(* IEC 61131-3 sources: AXOpen/src/components.rexroth.drives/ctrl/src/AxoCtrlxDriveXsc/v_6_x_x (part 3) *)

        ///<summary>
        /// This method  commands a controlled motion of a specified distance relative to the set position at the time of the execution.
        ///</summary>
        VAR INTERNAL
            MC_MoveRelativeExecute_PV					: 	BOOL;				//Execute - previous value
            MC_MoveRelativeErrorID					    : 	DINT;
            MC_MoveRelativeCycle					    : 	ULINT;
            MC_MoveRelativeContinuousUpdate_SV          :   BOOL;
            MC_MoveRelativeDistance_PV                  :   LREAL;
            MC_MoveRelativeVelocity_PV                  :   LREAL;
            MC_MoveRelativeAcceleration_PV              :   LREAL;
            MC_MoveRelativeDeceleration_PV              :   LREAL;
            MC_MoveRelativeJerk_PV                      :   LREAL;
        END_VAR
        METHOD PUBLIC OVERRIDE MC_MoveRelative
            VAR_INPUT
                AxisRef         :   AXOpen.Components.Abstractions.Drives.IAxoAxisReference;
                Execute         :   BOOL;                       //  Start the motion at rising edge
                ContinuousUpdate:   BOOL;                       //  Activate ‘ContinuousUpdate’ - target parameters should be changed during movement
                Distance        :   LREAL;                      //  Relative distance for the motion (in technical unit [u]
                Velocity        :   LREAL;                      //  Value of the maximum ‘Velocity’ (not necessarily reached) [u/s].
                Acceleration    :   LREAL;                      //  Value of the ‘Acceleration’ (always positive) (increasing energy of the motor) [u/s2]
                Deceleration    :   LREAL;                      //  Value of the ‘Deceleration’ (always positive) (decreasing energy of the motor) [u/s2]
                Jerk            :   LREAL;                      //  Value of the ‘Jerk’ [u/s3]
            END_VAR
            VAR_OUTPUT
                Done            :   BOOL;                       // Commanded distance reached
                Busy            :   BOOL;                       // The method is not finished and new output values are to be expected
                Active          :   BOOL;                       // Indicates that the method has control on the axis
                CommandAborted  :   BOOL;                       // ‘Command’ is aborted by another command
                Error           :   BOOL;                       // Signals that an error has occurred within the method
                ErrorID         :   DINT;                       // Error identification
            END_VAR
            VAR
                _AxisReference :  REF_TO AxoCtrlxDriveXscAxisReference;
            END_VAR

            _AxisReference ?= AxisRef;

            IF(_AxisReference = NULL) THEN
                Messenger.Activate(     UINT#1500, eAxoMessageCategory#ProgrammingError);
                DriveStatus.Error.Id := UINT#1500;
                RETURN;
            END_IF;

            IF THIS.AxoMoveRelative_Task.StartTriggered()  THEN
                _AxisReference^.Status.CurrentMotionTaskId := AXOpen.Components.Drives.eAxoMotionTaskId#Axo_MoveRelative;
            END_IF;

            IF Execute AND NOT MC_MoveRelativeExecute_PV AND _State = UINT#0 THEN
                _AxisReference^.Data.Cycle := _AxisReference^.Data.Cycle + ULINT#2;
                MC_MoveRelativeCycle := _AxisReference^.Data.Cycle ;
            END_IF;

            IF Execute THEN
                Messenger.ActivateOnCondition(ULINT#1501, Execute AND Velocity <= 0, eAxoMessageCategory#ProgrammingError);
                Messenger.ActivateOnCondition(ULINT#1502, Execute AND Acceleration <= 0, eAxoMessageCategory#ProgrammingError);
                Messenger.ActivateOnCondition(ULINT#1503, Execute AND Deceleration <= 0, eAxoMessageCategory#ProgrammingError);
                Messenger.ActivateOnCondition(ULINT#1504, Execute AND Jerk <= 0, eAxoMessageCategory#ProgrammingError);

                IF NOT ContinuousUpdate THEN
                    MC_MoveRelativeContinuousUpdate_SV := FALSE;
                END_IF;

                IF _State = UINT#0 THEN
                    Busy := TRUE;
                    Active := TRUE;
                    MC_MoveRelativeErrorID := DINT#0;
                    _AxisReference^.Outputs.SignalControlWord_S_0_0145_0_0.JogPositive := FALSE;
                    _AxisReference^.Outputs.SignalControlWord_S_0_0145_0_0.JogNegative := FALSE;
                    _AxisReference^.Outputs.SignalControlWord_S_0_0145_0_0.HomingControl:= FALSE;
                    _AxisReference^.Outputs.SignalControlWord_S_0_0145_0_0.AbsoluteRelative := TRUE;
                    _AxisReference^.Outputs.SignalControlWord_S_0_0145_0_0.ImmediateChange := TRUE;
                    MC_MoveRelativeContinuousUpdate_SV := ContinuousUpdate;
                    _State := UINT#360;
                    THIS.CallTimers(FALSE);
                END_IF;
                IF _State = UINT#360 THEN
                    IF _infoTimer.output THEN
                        TaskMessenger.Activate( UINT#560, eAxoMessageCategory#Potential);
                        DriveStatus.Error.Id := UINT#560;
                    END_IF;
                    Busy := TRUE;
                    Active := TRUE;
                    IF Velocity > 0 AND Acceleration > 0 AND Deceleration >0 AND Jerk > 0 THEN
                        _AxisReference^.Outputs.CommandPosition_S_0_0282_0_0 :=         TO_DINT(Distance        *   ScalingConstantRequiredPosition);
                        _AxisReference^.Outputs.CommandVelocity_S_0_0259_0_0 :=         TO_DINT(Velocity        *   ScalingConstantRequiredVelocity     * _AxisReference^.Data.OverrideVelocityFactor);
                        _AxisReference^.Outputs.CommandAcceleration_S_0_0260_0_0 :=     TO_DINT(Acceleration    *   ScalingConstantRequiredAcceleration * _AxisReference^.Data.OverrideAccelerationFactor);
                        _AxisReference^.Outputs.CommandDecceleration_S_0_0359_0_0 :=    TO_DINT(Deceleration    *   ScalingConstantRequiredDeceleration * _AxisReference^.Data.OverrideAccelerationFactor);
                        _AxisReference^.Outputs.CommandJerk_S_0_0193_0_0 :=             TO_DINT(Jerk            *   ScalingConstantRequiredJerk         * _AxisReference^.Data.OverrideJerkFactor);
                        MC_MoveRelativeDistance_PV      :=  Distance;
                        MC_MoveRelativeVelocity_PV      :=  Velocity;
                        MC_MoveRelativeAcceleration_PV  :=  Acceleration;
                        MC_MoveRelativeDeceleration_PV  :=  Deceleration;
                        MC_MoveRelativeJerk_PV          :=  Jerk;
                        _State := UINT#361;
                        THIS.CallTimers(FALSE);
                    END_IF;
                END_IF;
                IF _State = UINT#361 THEN
                    IF _infoTimer.output THEN
                        TaskMessenger.Activate( UINT#561, eAxoMessageCategory#Potential);
                        DriveStatus.Error.Id := UINT#561;
                    END_IF;
                    Busy := TRUE;
                    Active := TRUE;
                    _AxisReference^.Outputs.DriveControlWord_S_0_0134_0_0.CommandOperationModeBit0  := FALSE;
                    _AxisReference^.Outputs.DriveControlWord_S_0_0134_0_0.CommandOperationModeBit1  := FALSE;
                    _AxisReference^.Outputs.DriveControlWord_S_0_0134_0_0.CommandOperationModeBit2  := FALSE;
                    IF  NOT _AxisReference^.Inputs.DriveStatusWord_S_0_0135_0_0.ActualOperatingModeBit0 AND
                        NOT _AxisReference^.Inputs.DriveStatusWord_S_0_0135_0_0.ActualOperatingModeBit1 AND
                        NOT _AxisReference^.Inputs.DriveStatusWord_S_0_0135_0_0.ActualOperatingModeBit2 THEN
                        _State := UINT#362;
                        THIS.CallTimers(FALSE);
                    END_IF;
                END_IF;
                IF _State = UINT#362 THEN
                    IF _infoTimer.output THEN
                        TaskMessenger.Activate( UINT#562, eAxoMessageCategory#Potential);
                        DriveStatus.Error.Id := UINT#562;
                    END_IF;
                    Busy := TRUE;
                    Active := TRUE;
                    IF  _AxisReference^.Inputs.DriveStatusWord_S_0_0135_0_0.ReadyForOperationBit0 AND
                        _AxisReference^.Inputs.DriveStatusWord_S_0_0135_0_0.ReadyForOperationBit1 THEN
                       _State := UINT#363;
                        THIS.CallTimers(FALSE);
                    END_IF;
                END_IF;
                IF _State = UINT#363 THEN
                    IF _infoTimer.output THEN
                        TaskMessenger.Activate( UINT#563, eAxoMessageCategory#Potential);
                        DriveStatus.Error.Id := UINT#563;
                    END_IF;
                    Busy := TRUE;
                    Active := TRUE;
                    _AxisReference^.Outputs.DriveControlWord_S_0_0134_0_0.DriveHalt  := TRUE;
                    IF _AxisReference^.Inputs.DriveStatusWord_S_0_0135_0_0.CommandProcessingStatus AND NOT _AxisReference^.Inputs.DriveStatusWord_S_0_0135_0_0.InStandstill  THEN
                       _State := UINT#364;
                        THIS.CallTimers(FALSE);
                    END_IF;
                END_IF;
                //Executing movement
                IF _State = UINT#364 THEN
                    IF _infoTimer.output THEN
                        TaskMessenger.Activate( UINT#564, eAxoMessageCategory#Potential);
                        DriveStatus.Error.Id := UINT#564;
                    END_IF;
                    Busy := TRUE;
                    Active := TRUE;
                    _AxisReference^.Outputs.SignalControlWord_S_0_0145_0_0.AcceptanceOfPositioningCommandValue := NOT _AxisReference^.Outputs.SignalControlWord_S_0_0145_0_0.AcceptanceOfPositioningCommandValue; //_AxisReference^.Outputs.SignalControlWord_S_0_0145_0_0.AcceptanceOfPositioningCommandValue := NOT _AxisReference^.Inputs.SignalStatusWord_S_0_0144_0_0.PositionCommandAck;
                    IF TRUE THEN
                        _State := UINT#365;
                        THIS.CallTimers(FALSE);
                    END_IF;
                END_IF;
                IF _State = UINT#365 THEN
                    IF _infoTimer.output THEN
                        TaskMessenger.Activate( UINT#565, eAxoMessageCategory#Potential);
                        DriveStatus.Error.Id := UINT#565;
                    END_IF;
                    Busy := TRUE;
                    Active := TRUE;
                    IF _AxisReference^.Outputs.SignalControlWord_S_0_0145_0_0.AcceptanceOfPositioningCommandValue = _AxisReference^.Inputs.SignalStatusWord_S_0_0144_0_0.PositionCommandAck THEN
                        _State := UINT#366;
                        THIS.CallTimers(FALSE);
                    END_IF;
                END_IF;
                IF _State = UINT#366 THEN
                    IF _infoTimer.output THEN
                        TaskMessenger.Activate( UINT#566, eAxoMessageCategory#Potential);
                        DriveStatus.Error.Id := UINT#566;
                    END_IF;
                    IF _AxisReference^.Inputs.SignalStatusWord_S_0_0144_0_0.DriveStandstill AND _AxisReference^.Inputs.SignalStatusWord_S_0_0144_0_0.InTargetPosition THEN
                        _State := UINT#367;
                        THIS.CallTimers(FALSE);
                    END_IF;
                END_IF;
                IF _State = UINT#367 THEN
                    Done := TRUE;
                    MC_MoveRelativeCycle := ULINT#0;
                END_IF;
                IF _State = UINT#368 THEN
                    CommandAborted := TRUE; // action handled in parent AxoDrive
                END_IF;
                IF _State = UINT#369 THEN
                    MC_MoveRelativeCycle := ULINT#0;
                    Error := TRUE; // action handled in parent AxoDrive
                END_IF;

                IF _State>=UINT#360 AND _State<UINT#367 THEN
                    IF MC_MoveRelativeContinuousUpdate_SV AND (
                        MC_MoveRelativeDistance_PV      <>  Distance OR
                        MC_MoveRelativeVelocity_PV      <>  Velocity OR
                        MC_MoveRelativeAcceleration_PV  <>  Acceleration OR
                        MC_MoveRelativeDeceleration_PV  <>  Deceleration OR
                        MC_MoveRelativeJerk_PV          <>  Jerk ) THEN
                        IF TRUE THEN
                            _AxisReference^.Outputs.CommandPosition_S_0_0282_0_0 :=         TO_DINT(Distance        *   ScalingConstantRequiredPosition);
                            _AxisReference^.Outputs.CommandVelocity_S_0_0259_0_0 :=         TO_DINT(Velocity        *   ScalingConstantRequiredVelocity     * _AxisReference^.Data.OverrideVelocityFactor);
                            _AxisReference^.Outputs.CommandAcceleration_S_0_0260_0_0 :=     TO_DINT(Acceleration    *   ScalingConstantRequiredAcceleration * _AxisReference^.Data.OverrideAccelerationFactor);
                            _AxisReference^.Outputs.CommandDecceleration_S_0_0359_0_0 :=    TO_DINT(Deceleration    *   ScalingConstantRequiredDeceleration * _AxisReference^.Data.OverrideAccelerationFactor);
                            _AxisReference^.Outputs.CommandJerk_S_0_0193_0_0 :=             TO_DINT(Jerk            *   ScalingConstantRequiredJerk         * _AxisReference^.Data.OverrideJerkFactor);
                            MC_MoveRelativeDistance_PV      :=  Distance;
                            MC_MoveRelativeVelocity_PV      :=  Velocity;
                            MC_MoveRelativeAcceleration_PV  :=  Acceleration;
                            MC_MoveRelativeDeceleration_PV  :=  Deceleration;
                            MC_MoveRelativeJerk_PV          :=  Jerk;
                            _State := UINT#361;
                        END_IF;
                    END_IF;
                    IF NOT _AxisReference^.Inputs.DriveStatusWord_S_0_0135_0_0.ReadyForOperationBit0 OR NOT _AxisReference^.Inputs.DriveStatusWord_S_0_0135_0_0.ReadyForOperationBit1 THEN
                        _State := UINT#368;
                    ELSIF _AxisReference^.Inputs.DriveStatusWord_S_0_0135_0_0.DriveErrorZKL1 OR
                        (_AxisReference^.Inputs.DriveStatusWord_S_0_0135_0_0.WarningZKL2 AND _AxisReference^.Inputs.DiagnosticMessage_S_0_0390_0_0 >= DWORD#16#C00E0000) THEN
                        IF MC_MoveRelativeErrorID = DINT#0 THEN
                            MC_MoveRelativeErrorID := TO_DINT(_AxisReference^.Inputs.DiagnosticMessage_S_0_0390_0_0 AND DWORD#16#000FFFFF);
                        END_IF;
                        _State := UINT#369;
                    ELSIF _AxisReference^.Data.Cycle <> MC_MoveRelativeCycle THEN
                        _AxisReference^.Data.Cycle := _AxisReference^.Data.Cycle - ULINT#1;
                        _State := UINT#368;
                    END_IF;
                END_IF;

                THIS.CallTimers(TRUE,FALSE);
                THIS.AxoMoveRelative_Task.ThrowWhen(_errorTimer.output );
                THIS.AxoMoveRelative_Task.ThrowWhen(THIS.AxoMoveRelative_Task.Duration >= DriveConfig.TaskTimeout AND DriveConfig.TaskTimeout > T#0s ,'<#AxoMoveRelative_Task timeout.#>');
                DriveStatus.Action.Id := _State;
            END_IF;

            IF THIS.AxoMoveRelative_Task.DoneReached() AND _State>=UINT#360 AND _State<=UINT#369 THEN
                _AxisReference^.Status.CurrentMotionTaskId := AXOpen.Components.Drives.eAxoMotionTaskId#Axo_Done;
                MC_MoveRelativeErrorID := DINT#0;
                // MC_MoveRelativeCycle := ULINT#0;
                _State := UINT#0;
            END_IF;

            IF THIS.AxoMoveRelative_Task.RestoreTriggered() AND _State>=UINT#360 AND _State<=UINT#369 THEN
                _AxisReference^.Status.CurrentMotionTaskId := AXOpen.Components.Drives.eAxoMotionTaskId#Axo_None;
                MC_MoveRelativeErrorID := DINT#0;
                MC_MoveRelativeCycle := ULINT#0;
                _State := UINT#0;
            END_IF;
            ErrorID := MC_MoveRelativeErrorID;
            MC_MoveRelativeExecute_PV := Execute;
        END_METHOD

        ///<summary>
        /// This method commands a controlled motion of a specified relative distance additional to the most recent
        /// commanded position in the axis_State ‘DiscreteMotion’. The most recent commanded position may be the result of a
        /// previous MC_MoveAdditive motion which was aborted. If the method is activated in the axis_State ‘ContinuousMotion’, the
        /// specified relative distance is added to the set position at the time of the execution.
        ///</summary>
        VAR INTERNAL
            MC_MoveAdditiveExecute_PV					: 	BOOL;				//Execute - previous value
            MC_MoveAdditiveErrorID					    : 	DINT;
            MC_MoveAdditiveCycle					    : 	ULINT;
            MC_MoveAdditiveContinuousUpdate_SV          :   BOOL;
            MC_MoveAdditiveDistance_PV                  :   LREAL;
            MC_MoveAdditiveVelocity_PV                  :   LREAL;
            MC_MoveAdditiveAcceleration_PV              :   LREAL;
            MC_MoveAdditiveDeceleration_PV              :   LREAL;
            MC_MoveAdditiveJerk_PV                      :   LREAL;
        END_VAR
        METHOD PUBLIC OVERRIDE MC_MoveAdditive
            VAR_INPUT
                AxisRef         :   AXOpen.Components.Abstractions.Drives.IAxoAxisReference;
                Execute         :   BOOL;                       //  Start the motion at rising edge
                ContinuousUpdate:   BOOL;                       //  Activate ‘ContinuousUpdate’ - target parameters should be changed during movement
                Distance        :   LREAL;                      //  Relative distance for the motion (in technical unit [u]
                Velocity        :   LREAL;                      //  Value of the maximum ‘Velocity’ (not necessarily reached) [u/s].
                Acceleration    :   LREAL;                      //  Value of the ‘Acceleration’ (always positive) (increasing energy of the motor) [u/s2]
                Deceleration    :   LREAL;                      //  Value of the ‘Deceleration’ (always positive) (decreasing energy of the motor) [u/s2]
                Jerk            :   LREAL;                      //  Value of the ‘Jerk’ [u/s3]
            END_VAR
            VAR_OUTPUT
                Done            :   BOOL;                       // Commanded distance reached
                Busy            :   BOOL;                       // The method is not finished and new output values are to be expected
                Active          :   BOOL;                       // Indicates that the method has control on the axis
                CommandAborted  :   BOOL;                       // ‘Command’ is aborted by another command
                Error           :   BOOL;                       // Signals that an error has occurred within the method
                ErrorID         :   DINT;                       // Error identification
            END_VAR
            VAR
                _AxisReference :  REF_TO AxoCtrlxDriveXscAxisReference;
            END_VAR

            _AxisReference ?= AxisRef;

            IF(_AxisReference = NULL) THEN
                Messenger.Activate(     UINT#1510, eAxoMessageCategory#ProgrammingError);
                DriveStatus.Error.Id := UINT#1510;
                RETURN;
            END_IF;

            IF Execute AND NOT MC_MoveAdditiveExecute_PV THEN
                _State := UINT#0;  //TODO check if this casues the issue with two move relative movements???
            END_IF;

            IF Execute THEN
                Messenger.ActivateOnCondition(ULINT#1511, Execute AND Velocity <= 0, eAxoMessageCategory#ProgrammingError);
                Messenger.ActivateOnCondition(ULINT#1512, Execute AND Acceleration <= 0, eAxoMessageCategory#ProgrammingError);
                Messenger.ActivateOnCondition(ULINT#1513, Execute AND Deceleration <= 0, eAxoMessageCategory#ProgrammingError);
                Messenger.ActivateOnCondition(ULINT#1514, Execute AND Jerk <= 0, eAxoMessageCategory#ProgrammingError);

                IF NOT ContinuousUpdate THEN
                    MC_MoveAdditiveContinuousUpdate_SV := FALSE;
                END_IF;

                IF _State = UINT#0 THEN
                    Busy := TRUE;
                    Active := TRUE;
                    MC_MoveAdditiveErrorID := DINT#0;
                    _AxisReference^.Outputs.SignalControlWord_S_0_0145_0_0.JogPositive := FALSE;
                    _AxisReference^.Outputs.SignalControlWord_S_0_0145_0_0.JogNegative := FALSE;
                    _AxisReference^.Outputs.SignalControlWord_S_0_0145_0_0.HomingControl:= FALSE;
                    _AxisReference^.Outputs.SignalControlWord_S_0_0145_0_0.ImmediateChange := TRUE;
                    MC_MoveAdditiveContinuousUpdate_SV := ContinuousUpdate;
                    IF Velocity > 0 AND Acceleration > 0 AND Deceleration >0 AND Jerk > 0 THEN
                        MC_MoveAdditiveDistance_PV      :=  Distance;
                        MC_MoveAdditiveVelocity_PV      :=  Velocity;
                        MC_MoveAdditiveAcceleration_PV  :=  Acceleration;
                        MC_MoveAdditiveDeceleration_PV  :=  Deceleration;
                        MC_MoveAdditiveJerk_PV          :=  Jerk;
                        IF _AxisReference^.Status.CurrentMotionTaskId = eAxoMotionTaskId#Axo_MoveAbsolute THEN
                            AxoMoveAbsolute_Task.Abort();
                            _AxisReference^.Outputs.SignalControlWord_S_0_0145_0_0.AbsoluteRelative := FALSE;
                            _AxisReference^.Outputs.CommandPosition_S_0_0282_0_0 :=         TO_DINT((MC_MoveAbsolutePosition_PV + Distance) * ScalingConstantRequiredPosition);
                            _AxisReference^.Outputs.CommandVelocity_S_0_0259_0_0 :=         TO_DINT(Velocity        *   ScalingConstantRequiredVelocity         * _AxisReference^.Data.OverrideVelocityFactor);
                            _AxisReference^.Outputs.CommandAcceleration_S_0_0260_0_0 :=     TO_UINT(Acceleration    *   ScalingConstantRequiredAcceleration     * _AxisReference^.Data.OverrideAccelerationFactor);
                            _AxisReference^.Outputs.CommandDecceleration_S_0_0359_0_0 :=    TO_UINT(Deceleration    *   ScalingConstantRequiredDeceleration     * _AxisReference^.Data.OverrideAccelerationFactor);
                            _AxisReference^.Outputs.CommandJerk_S_0_0193_0_0 :=             TO_DINT(Jerk            *   ScalingConstantRequiredJerk             * _AxisReference^.Data.OverrideJerkFactor);
                        ELSE
                            _AxisReference^.Outputs.SignalControlWord_S_0_0145_0_0.AbsoluteRelative := TRUE;
                            _AxisReference^.Outputs.CommandPosition_S_0_0282_0_0 :=         TO_DINT((Distance)      *   ScalingConstantRequiredPosition);
                            _AxisReference^.Outputs.CommandVelocity_S_0_0259_0_0 :=         TO_DINT(Velocity        *   ScalingConstantRequiredVelocity         * _AxisReference^.Data.OverrideVelocityFactor);
                            _AxisReference^.Outputs.CommandAcceleration_S_0_0260_0_0 :=     TO_UINT(Acceleration    *   ScalingConstantRequiredAcceleration     * _AxisReference^.Data.OverrideAccelerationFactor);
                            _AxisReference^.Outputs.CommandDecceleration_S_0_0359_0_0 :=    TO_UINT(Deceleration    *   ScalingConstantRequiredDeceleration     * _AxisReference^.Data.OverrideAccelerationFactor);
                            _AxisReference^.Outputs.CommandJerk_S_0_0193_0_0 :=             TO_DINT(Jerk            *   ScalingConstantRequiredJerk             * _AxisReference^.Data.OverrideJerkFactor);
                        END_IF;
                        IF _AxisReference^.Status.CurrentMotionTaskId = eAxoMotionTaskId#Axo_MoveRelative THEN
                            AxoMoveRelative_Task.Abort();
                        END_IF;
                        _AxisReference^.Status.CurrentMotionTaskId := eAxoMotionTaskId#Axo_MoveAdditive;
                        _AxisReference^.Data.Cycle := _AxisReference^.Data.Cycle + ULINT#2;
                        MC_MoveAdditiveCycle := _AxisReference^.Data.Cycle ;
                        _State := UINT#371;
                        THIS.CallTimers(FALSE);
                    END_IF;
                END_IF;
                IF _State = UINT#370 THEN
                    _State := UINT#371;
                    THIS.CallTimers(FALSE);
                END_IF;
                IF _State = UINT#371 THEN
                    IF _infoTimer.output THEN
                        TaskMessenger.Activate( UINT#571, eAxoMessageCategory#Potential);
                        DriveStatus.Error.Id := UINT#571;
                    END_IF;
                    Busy := TRUE;
                    Active := TRUE;
                    _AxisReference^.Outputs.DriveControlWord_S_0_0134_0_0.CommandOperationModeBit0  := FALSE;
                    _AxisReference^.Outputs.DriveControlWord_S_0_0134_0_0.CommandOperationModeBit1  := FALSE;
                    _AxisReference^.Outputs.DriveControlWord_S_0_0134_0_0.CommandOperationModeBit2  := FALSE;
                    IF  NOT _AxisReference^.Inputs.DriveStatusWord_S_0_0135_0_0.ActualOperatingModeBit0 AND
                        NOT _AxisReference^.Inputs.DriveStatusWord_S_0_0135_0_0.ActualOperatingModeBit1 AND
                        NOT _AxisReference^.Inputs.DriveStatusWord_S_0_0135_0_0.ActualOperatingModeBit2 THEN
                        _State := UINT#372;
                        THIS.CallTimers(FALSE);
                    END_IF;
                END_IF;
                IF _State = UINT#372 THEN
                    IF _infoTimer.output THEN
                        TaskMessenger.Activate( UINT#572, eAxoMessageCategory#Potential);
                        DriveStatus.Error.Id := UINT#572;
                    END_IF;
                    Busy := TRUE;
                    Active := TRUE;
                    IF  _AxisReference^.Inputs.DriveStatusWord_S_0_0135_0_0.ReadyForOperationBit0 AND
                        _AxisReference^.Inputs.DriveStatusWord_S_0_0135_0_0.ReadyForOperationBit1 THEN
                       _State := UINT#373;
                        THIS.CallTimers(FALSE);
                    END_IF;
                END_IF;
                IF _State = UINT#373 THEN
                    IF _infoTimer.output THEN
                        TaskMessenger.Activate( UINT#573, eAxoMessageCategory#Potential);
                        DriveStatus.Error.Id := UINT#573;
                    END_IF;
                    Busy := TRUE;
                    Active := TRUE;
                    _AxisReference^.Outputs.DriveControlWord_S_0_0134_0_0.DriveHalt  := TRUE;
                    IF _AxisReference^.Inputs.DriveStatusWord_S_0_0135_0_0.CommandProcessingStatus AND NOT _AxisReference^.Inputs.DriveStatusWord_S_0_0135_0_0.InStandstill  THEN
                       _State := UINT#374;
                        THIS.CallTimers(FALSE);
                    END_IF;
                END_IF;
                IF _State = UINT#374 THEN
                    IF _infoTimer.output THEN
                        TaskMessenger.Activate( UINT#574, eAxoMessageCategory#Potential);
                        DriveStatus.Error.Id := UINT#574;
                    END_IF;
                    Busy := TRUE;
                    Active := TRUE;
                    _AxisReference^.Outputs.SignalControlWord_S_0_0145_0_0.AcceptanceOfPositioningCommandValue := NOT _AxisReference^.Outputs.SignalControlWord_S_0_0145_0_0.AcceptanceOfPositioningCommandValue; //_AxisReference^.Outputs.SignalControlWord_S_0_0145_0_0.AcceptanceOfPositioningCommandValue := NOT _AxisReference^.Inputs.SignalStatusWord_S_0_0144_0_0.PositionCommandAck;
                    IF TRUE THEN
                        _State := UINT#375;
                        THIS.CallTimers(FALSE);
                    END_IF;
                END_IF;
                IF _State = UINT#375 THEN
                    IF _infoTimer.output THEN
                        TaskMessenger.Activate( UINT#575, eAxoMessageCategory#Potential);
                        DriveStatus.Error.Id := UINT#575;
                    END_IF;
                    Busy := TRUE;
                    Active := TRUE;
                    IF _AxisReference^.Outputs.SignalControlWord_S_0_0145_0_0.AcceptanceOfPositioningCommandValue = _AxisReference^.Inputs.SignalStatusWord_S_0_0144_0_0.PositionCommandAck THEN
                        _State := UINT#376;
                        THIS.CallTimers(FALSE);
                    END_IF;
                END_IF;
                IF _State = UINT#376 THEN
                    IF _infoTimer.output THEN
                        TaskMessenger.Activate( UINT#576, eAxoMessageCategory#Potential);
                        DriveStatus.Error.Id := UINT#576;
                    END_IF;
                    IF _AxisReference^.Inputs.SignalStatusWord_S_0_0144_0_0.DriveStandstill AND _AxisReference^.Inputs.SignalStatusWord_S_0_0144_0_0.InTargetPosition THEN
                        _State := UINT#377;
                        THIS.CallTimers(FALSE);
                    END_IF;
                END_IF;
                IF _State = UINT#377 THEN
                    Done := TRUE;
                    MC_MoveAdditiveCycle := ULINT#0;
                END_IF;
                IF _State = UINT#378 THEN
                    CommandAborted := TRUE; // action handled in parent AxoDrive
                END_IF;
                IF _State = UINT#379 THEN
                    MC_MoveAdditiveCycle := ULINT#0;
                    Error := TRUE; // action handled in parent AxoDrive
                END_IF;

                IF _State>=UINT#370 AND _State<UINT#377 THEN
                    IF MC_MoveAdditiveContinuousUpdate_SV AND (
                        MC_MoveAdditiveDistance_PV      <>  Distance OR
                        MC_MoveAdditiveVelocity_PV      <>  Velocity OR
                        MC_MoveAdditiveAcceleration_PV  <>  Acceleration OR
                        MC_MoveAdditiveDeceleration_PV  <>  Deceleration OR
                        MC_MoveAdditiveJerk_PV          <>  Jerk ) THEN
                        IF TRUE THEN
                            IF NOT _AxisReference^.Outputs.SignalControlWord_S_0_0145_0_0.AbsoluteRelative THEN
                                _AxisReference^.Outputs.CommandPosition_S_0_0282_0_0 :=_AxisReference^.Outputs.CommandPosition_S_0_0282_0_0  + TO_DINT((Distance - MC_MoveAdditiveDistance_PV) * ScalingConstantRequiredPosition);
                            ELSE
                                _AxisReference^.Outputs.CommandPosition_S_0_0282_0_0 := TO_DINT((Distance) * ScalingConstantRequiredPosition) - _AxisReference^.Inputs.ActualPosition_S_0_0386_0_0;
                            END_IF;
                            _AxisReference^.Outputs.CommandVelocity_S_0_0259_0_0 :=         TO_DINT(Velocity        *   ScalingConstantRequiredVelocity     * _AxisReference^.Data.OverrideVelocityFactor);
                            _AxisReference^.Outputs.CommandAcceleration_S_0_0260_0_0 :=     TO_UINT(Acceleration    *   ScalingConstantRequiredAcceleration * _AxisReference^.Data.OverrideAccelerationFactor);
                            _AxisReference^.Outputs.CommandDecceleration_S_0_0359_0_0 :=    TO_UINT(Deceleration    *   ScalingConstantRequiredDeceleration * _AxisReference^.Data.OverrideAccelerationFactor);
                            _AxisReference^.Outputs.CommandJerk_S_0_0193_0_0 :=             TO_UINT(Jerk            *   ScalingConstantRequiredJerk         * _AxisReference^.Data.OverrideJerkFactor);
                            MC_MoveAdditiveDistance_PV      :=  Distance;
                            MC_MoveAdditiveVelocity_PV      :=  Velocity;
                            MC_MoveAdditiveAcceleration_PV  :=  Acceleration;
                            MC_MoveAdditiveDeceleration_PV  :=  Deceleration;
                            MC_MoveAdditiveJerk_PV          :=  Jerk;
                            _State := UINT#371;
                        END_IF;
                    END_IF;
                    IF NOT _AxisReference^.Inputs.DriveStatusWord_S_0_0135_0_0.ReadyForOperationBit0 OR NOT _AxisReference^.Inputs.DriveStatusWord_S_0_0135_0_0.ReadyForOperationBit1 THEN
                        _State := UINT#378;
                    ELSIF _AxisReference^.Inputs.DriveStatusWord_S_0_0135_0_0.DriveErrorZKL1 OR
                        (_AxisReference^.Inputs.DriveStatusWord_S_0_0135_0_0.WarningZKL2 AND _AxisReference^.Inputs.DiagnosticMessage_S_0_0390_0_0 >= DWORD#16#C00E0000) THEN
                        IF MC_MoveAdditiveErrorID = DINT#0 THEN
                            MC_MoveAdditiveErrorID := TO_DINT(_AxisReference^.Inputs.DiagnosticMessage_S_0_0390_0_0 AND DWORD#16#000FFFFF);
                        END_IF;
                        _State := UINT#379;
                    ELSIF _AxisReference^.Data.Cycle <> MC_MoveAdditiveCycle THEN
                        _AxisReference^.Data.Cycle := _AxisReference^.Data.Cycle - ULINT#1;
                        _State := UINT#378;
                    END_IF;
                END_IF;
                THIS.CallTimers(TRUE,FALSE);
                THIS.AxoMoveAdditive_Task.ThrowWhen(_errorTimer.output );
                THIS.AxoMoveAdditive_Task.ThrowWhen(THIS.AxoMoveAdditive_Task.Duration >= DriveConfig.TaskTimeout AND DriveConfig.TaskTimeout > T#0s ,'<#AxoMoveAdditive_Task timeout.#>');
                DriveStatus.Action.Id := _State;
            END_IF;

            IF THIS.AxoMoveAdditive_Task.DoneReached() AND _State>=UINT#370 AND _State<=UINT#379 THEN
                _AxisReference^.Status.CurrentMotionTaskId := AXOpen.Components.Drives.eAxoMotionTaskId#Axo_Done;
                MC_MoveAdditiveErrorID := DINT#0;
                // MC_MoveAdditiveCycle := ULINT#0;
                _State := UINT#0;
            END_IF;

            IF THIS.AxoMoveAdditive_Task.RestoreTriggered() AND _State>=UINT#370 AND _State<=UINT#379 THEN
                _AxisReference^.Status.CurrentMotionTaskId := AXOpen.Components.Drives.eAxoMotionTaskId#Axo_None;
                MC_MoveAdditiveErrorID := DINT#0;
                MC_MoveAdditiveCycle := ULINT#0;
                _State := UINT#0;
            END_IF;

            ErrorID := MC_MoveAdditiveErrorID;
            MC_MoveAdditiveExecute_PV := Execute;
        END_METHOD

        ///<summary>
        /// This method commands a never ending controlled motion at a specified velocity.
        ///</summary>
        VAR INTERNAL
            MC_MoveVelocityExecute_PV					: 	BOOL;				//Execute - previous value
            MC_MoveVelocityErrorID					    : 	DINT;
            MC_MoveVelocityCycle					    : 	ULINT;
            MC_MoveVelocityContinuousUpdate_SV          :   BOOL;
            MC_MoveVelocityVelocity_PV                  :   LREAL;
            MC_MoveVelocityAcceleration_PV              :   LREAL;
            MC_MoveVelocityDeceleration_PV              :   LREAL;
            MC_MoveVelocityJerk_PV                      :   LREAL;
            MC_MoveVelocityDirection_PV                 :   AXOpen.Components.Abstractions.Drives.eAxoDriveDirection;
        END_VAR
        METHOD PUBLIC OVERRIDE MC_MoveVelocity
            VAR_INPUT
                AxisRef         :   AXOpen.Components.Abstractions.Drives.IAxoAxisReference;
                Execute         :   BOOL;                       //  Start the motion at rising edge
                ContinuousUpdate:   BOOL;                       //  Activate ‘ContinuousUpdate’ - target parameters should be changed during movement
                Velocity        :   LREAL;                      //  Value of the maximum velocity [u/s]. Can be a signed value.
                Acceleration    :   LREAL;                      //  Value of the ‘Acceleration’ (always positive) (increasing energy of the motor) [u/s2]
                Deceleration    :   LREAL;                      //  Value of the ‘Deceleration’ (always positive) (decreasing energy of the motor) [u/s2]
                Jerk            :   LREAL;                      //  Value of the ‘Jerk’ [u/s3]
                Direction       :   AXOpen.Components.Abstractions.Drives.eAxoDriveDirection;         //  Enum type (1-of-3 values: PositiveDirection, NegativeDirection, and CurrentDirection. Note: shortest way not applicable)
            END_VAR
            VAR_OUTPUT
                InVelocity      :   BOOL;                       // Commanded velocity reached
                Busy            :   BOOL;                       // The method is not finished and new output values are to be expected
                Active          :   BOOL;                       // Indicates that the method has control on the axis
                CommandAborted  :   BOOL;                       // ‘Command’ is aborted by another command
                Error           :   BOOL;                       // Signals that an error has occurred within the method
                ErrorID         :   DINT;                       // Error identification
            END_VAR
            VAR
                _AxisReference :  REF_TO AxoCtrlxDriveXscAxisReference;
                Velocity_   :   LREAL;
                Direction_  :   AXOpen.Components.Abstractions.Drives.eAxoDriveDirection;
                VelocityWindowPerCent     :   LREAL := LREAL#5.0;
                VelocityWindowMin         :   LREAL;
                VelocityWindowMax         :   LREAL;
            END_VAR

            _AxisReference ?= AxisRef;

            IF(_AxisReference = NULL) THEN
                Messenger.Activate(     UINT#1520, eAxoMessageCategory#ProgrammingError);
                DriveStatus.Error.Id := UINT#1520;
                RETURN;
            END_IF;

            IF THIS.AxoMoveVelocity_Task.StartTriggered()  THEN
                _AxisReference^.Status.CurrentMotionTaskId := AXOpen.Components.Drives.eAxoMotionTaskId#Axo_MoveVelocity;
            END_IF;

            IF Execute AND NOT MC_MoveVelocityExecute_PV AND _State = UINT#0 THEN
                _AxisReference^.Data.Cycle := _AxisReference^.Data.Cycle + ULINT#2;
                MC_MoveVelocityCycle := _AxisReference^.Data.Cycle ;
            END_IF;

            IF Execute THEN
                Messenger.ActivateOnCondition(ULINT#1521,Direction <> AXOpen.Components.Abstractions.Drives.eAxoDriveDirection#PositiveDirection AND Direction <> AXOpen.Components.Abstractions.Drives.eAxoDriveDirection#NegativeDirection, eAxoMessageCategory#ProgrammingError);

                IF Direction = AXOpen.Components.Abstractions.Drives.eAxoDriveDirection#PositiveDirection THEN
                    Velocity_ := Velocity;
                ELSIF Direction = AXOpen.Components.Abstractions.Drives.eAxoDriveDirection#NegativeDirection THEN
                    Velocity_ := -1 * Velocity;
                ELSE
                    RETURN;
                END_IF;

                IF Velocity_> 0 THEN
                    Direction_ := AXOpen.Components.Abstractions.Drives.eAxoDriveDirection#PositiveDirection;
                ELSE
                    Direction_ := AXOpen.Components.Abstractions.Drives.eAxoDriveDirection#NegativeDirection;
                END_IF;

                Messenger.ActivateOnCondition(ULINT#1522, Execute AND Velocity = 0, eAxoMessageCategory#ProgrammingError);
                Messenger.ActivateOnCondition(ULINT#1523, Execute AND Acceleration <= 0, eAxoMessageCategory#ProgrammingError);
                Messenger.ActivateOnCondition(ULINT#1524, Execute AND Deceleration <= 0, eAxoMessageCategory#ProgrammingError);
                Messenger.ActivateOnCondition(ULINT#1525, Execute AND Jerk <= 0, eAxoMessageCategory#ProgrammingError);

                IF NOT ContinuousUpdate THEN
                    MC_MoveVelocityContinuousUpdate_SV := FALSE;
                END_IF;

                IF _State = UINT#0 THEN
                    Busy    := TRUE;
                    Active  := TRUE;
                    MC_MoveVelocityErrorID := DINT#0;
                    _AxisReference^.Outputs.DriveControlWord_S_0_0134_0_0.CommandOperationModeBit0 := FALSE;
                    _AxisReference^.Outputs.DriveControlWord_S_0_0134_0_0.CommandOperationModeBit1 := FALSE;
                    _AxisReference^.Outputs.DriveControlWord_S_0_0134_0_0.CommandOperationModeBit2 := FALSE;
                    // _AxisReference^.Outputs.DriveControlWord_S_0_0134_0_0.DriveHalt := FALSE;
                    // _AxisReference^.Outputs.DriveControlWord_S_0_0134_0_0.DriveEnable := FALSE;
                    // _AxisReference^.Outputs.DriveControlWord_S_0_0134_0_0.DriveOn := FALSE;
                    // _AxisReference^.Outputs.SignalControlWord_S_0_0145_0_0.AcceptanceOfPositioningCommandValue := FALSE;
                    _AxisReference^.Outputs.SignalControlWord_S_0_0145_0_0.HomingControl := FALSE;
                    _AxisReference^.Outputs.SignalControlWord_S_0_0145_0_0.AbsoluteRelative := FALSE;
                    _AxisReference^.Outputs.SignalControlWord_S_0_0145_0_0.ImmediateChange := FALSE;
                    _AxisReference^.Outputs.SignalControlWord_S_0_0145_0_0.ClearError := FALSE;
                    _AxisReference^.Outputs.SignalControlWord_S_0_0145_0_0.JogPositive := FALSE;
                    _AxisReference^.Outputs.SignalControlWord_S_0_0145_0_0.JogNegative := FALSE;
                    _AxisReference^.Outputs.SignalControlWord_S_0_0145_0_0.SwitchToCM := FALSE;
                    _AxisReference^.Outputs.SignalControlWord_S_0_0145_0_0.SwitchTo0M := TRUE;
                    // _AxisReference^.Outputs.SignalControlWord_S_0_0145_0_0.CancelReferencePoint := FALSE;
                    // _AxisReference^.Outputs.SignalControlWord_S_0_0145_0_0.SetAbsPositionFunction := FALSE;

                    MC_MoveVelocityContinuousUpdate_SV := ContinuousUpdate;
                    _State := UINT#380;
                    THIS.CallTimers(FALSE);
                END_IF;
                IF _State = UINT#380 THEN
                    Busy := TRUE;
                    Active := TRUE;
                    IF Velocity <> 0 AND Acceleration > 0 AND Deceleration >0 AND Jerk > 0 THEN
                        _AxisReference^.Outputs.CommandPosition_S_0_0282_0_0        :=  TO_DINT(0.0             *   ScalingConstantRequiredPosition);
                        _AxisReference^.Outputs.CommandVelocity_S_0_0259_0_0        :=  TO_DINT(Velocity_       *   ScalingConstantRequiredVelocity     *   _AxisReference^.Data.OverrideVelocityFactor);
                        _AxisReference^.Outputs.CommandAcceleration_S_0_0260_0_0    :=  TO_DINT(Acceleration    *   ScalingConstantRequiredAcceleration *   _AxisReference^.Data.OverrideAccelerationFactor);
                        _AxisReference^.Outputs.CommandDecceleration_S_0_0359_0_0   :=  TO_DINT(Deceleration    *   ScalingConstantRequiredDeceleration *   _AxisReference^.Data.OverrideAccelerationFactor);
                        _AxisReference^.Outputs.CommandJerk_S_0_0193_0_0            :=  TO_DINT(Jerk            *   ScalingConstantRequiredJerk         *   _AxisReference^.Data.OverrideJerkFactor);

                        MC_MoveVelocityVelocity_PV      :=  Velocity_;
                        MC_MoveVelocityAcceleration_PV  :=  Acceleration;
                        MC_MoveVelocityDeceleration_PV  :=  Deceleration;
                        MC_MoveVelocityJerk_PV          :=  Jerk;
                        MC_MoveVelocityDirection_PV     :=  Direction_;
                        _State := UINT#381;
                        THIS.CallTimers(FALSE);
                    END_IF;
                END_IF;
                IF _State = UINT#381 THEN
                    IF _infoTimer.output THEN
                        TaskMessenger.Activate( UINT#581, eAxoMessageCategory#Potential);
                        DriveStatus.Error.Id := UINT#581;
                    END_IF;
                    Busy := TRUE;
                    Active := TRUE;
                    _AxisReference^.Outputs.DriveControlWord_S_0_0134_0_0.CommandOperationModeBit0  := FALSE;
                    _AxisReference^.Outputs.DriveControlWord_S_0_0134_0_0.CommandOperationModeBit1  := FALSE;
                    _AxisReference^.Outputs.DriveControlWord_S_0_0134_0_0.CommandOperationModeBit2  := FALSE;
                    IF  NOT _AxisReference^.Inputs.DriveStatusWord_S_0_0135_0_0.ActualOperatingModeBit0 AND
                        NOT _AxisReference^.Inputs.DriveStatusWord_S_0_0135_0_0.ActualOperatingModeBit1 AND
                        NOT _AxisReference^.Inputs.DriveStatusWord_S_0_0135_0_0.ActualOperatingModeBit2 THEN
                        _State := UINT#382;
                        THIS.CallTimers(FALSE);
                    END_IF;
                END_IF;
                IF _State = UINT#382 THEN
                    IF _infoTimer.output THEN
                        TaskMessenger.Activate( UINT#582, eAxoMessageCategory#Potential);
                        DriveStatus.Error.Id := UINT#582;
                    END_IF;
                    Busy := TRUE;
                    Active := TRUE;
                    IF  _AxisReference^.Inputs.DriveStatusWord_S_0_0135_0_0.ReadyForOperationBit0 AND
                        _AxisReference^.Inputs.DriveStatusWord_S_0_0135_0_0.ReadyForOperationBit1 THEN
                       _State := UINT#383;
                        THIS.CallTimers(FALSE);
                    END_IF;
                END_IF;
                IF _State = UINT#383 THEN
                    IF _infoTimer.output THEN
                        TaskMessenger.Activate( UINT#583, eAxoMessageCategory#Potential);
                        DriveStatus.Error.Id := UINT#583;
                    END_IF;
                    Busy := TRUE;
                    Active := TRUE;
                    _AxisReference^.Outputs.DriveControlWord_S_0_0134_0_0.DriveHalt := TRUE;
                    IF _AxisReference^.Inputs.DriveStatusWord_S_0_0135_0_0.CommandProcessingStatus AND NOT _AxisReference^.Inputs.DriveStatusWord_S_0_0135_0_0.InStandstill  THEN
                        _State := UINT#384;
                        THIS.CallTimers(FALSE);
                    END_IF;
                END_IF;
                IF _State = UINT#384 THEN
                    IF _infoTimer.output THEN
                        TaskMessenger.Activate( UINT#584, eAxoMessageCategory#Potential);
                        DriveStatus.Error.Id := UINT#584;
                    END_IF;
                    Busy := TRUE;
                    Active := TRUE;
                    IF Direction_ = AXOpen.Components.Abstractions.Drives.eAxoDriveDirection#PositiveDirection THEN
                        _AxisReference^.Outputs.SignalControlWord_S_0_0145_0_0.JogPositive := TRUE;
                        _AxisReference^.Outputs.SignalControlWord_S_0_0145_0_0.JogNegative := FALSE;
                    ELSIF Direction_ = AXOpen.Components.Abstractions.Drives.eAxoDriveDirection#NegativeDirection THEN
                        _AxisReference^.Outputs.SignalControlWord_S_0_0145_0_0.JogPositive := FALSE;
                        _AxisReference^.Outputs.SignalControlWord_S_0_0145_0_0.JogNegative := TRUE;
                    END_IF;

                    IF NOT _AxisReference^.Inputs.DriveStatusWord_S_0_0135_0_0.InStandstill THEN
                        _State := UINT#385;
                        THIS.CallTimers(FALSE);
                    END_IF;
                END_IF;
                IF _State = UINT#385 THEN
                    IF TRUE THEN
                        _State := UINT#386;
                        THIS.CallTimers(FALSE);
                    END_IF;
                END_IF;
                IF Direction_ = AXOpen.Components.Abstractions.Drives.eAxoDriveDirection#PositiveDirection  THEN
                    VelocityWindowMax := Velocity_ + (Velocity_ * VelocityWindowPerCent / REAL#100.0);
                    VelocityWindowMin := Velocity_ - (Velocity_ * VelocityWindowPerCent / REAL#100.0);
                ELSE
                    VelocityWindowMax := Velocity_ - (Velocity_ * VelocityWindowPerCent / REAL#100.0);
                    VelocityWindowMin := Velocity_ + (Velocity_ * VelocityWindowPerCent / REAL#100.0);
                END_IF;
                InVelocity := ActualVelocity >= VelocityWindowMin AND ActualVelocity <= VelocityWindowMax;
                IF _State = UINT#386 THEN
                    IF _infoTimer.output THEN
                        TaskMessenger.Activate( UINT#586, eAxoMessageCategory#Potential);
                        DriveStatus.Error.Id := UINT#586;
                    END_IF;
                    IF InVelocity AND NOT MC_MoveVelocityContinuousUpdate_SV THEN
                        _State := UINT#387;
                        THIS.CallTimers(FALSE);
                    END_IF;
                END_IF;
                IF _State = UINT#387 THEN
                    MC_MoveVelocityCycle := ULINT#0;
                END_IF;
                IF _State = UINT#388 THEN
                    _AxisReference^.Outputs.SignalControlWord_S_0_0145_0_0.JogPositive := FALSE;
                    _AxisReference^.Outputs.SignalControlWord_S_0_0145_0_0.JogNegative := FALSE;
                    CommandAborted := TRUE; // action handled in parent AxoDrive
                END_IF;
                IF _State = UINT#389 THEN
                    _AxisReference^.Outputs.SignalControlWord_S_0_0145_0_0.JogPositive := FALSE;
                    _AxisReference^.Outputs.SignalControlWord_S_0_0145_0_0.JogNegative := FALSE;
                    MC_MoveVelocityCycle := ULINT#0;
                    Error := TRUE; // action handled in parent AxoDrive
                END_IF;

                IF _State>=UINT#380 AND _State<UINT#387 THEN
                    IF MC_MoveVelocityContinuousUpdate_SV AND (
                        MC_MoveVelocityVelocity_PV      <>  Velocity_ OR
                        MC_MoveVelocityAcceleration_PV  <>  Acceleration OR
                        MC_MoveVelocityDeceleration_PV  <>  Deceleration OR
                        MC_MoveVelocityJerk_PV          <>  Jerk OR
                        MC_MoveVelocityDirection_PV     <>  Direction_ ) THEN
                        IF TRUE THEN
                            _AxisReference^.Outputs.SignalControlWord_S_0_0145_0_0.ImmediateChange := TRUE;
                            _State := UINT#380;
                        END_IF;
                    END_IF;
                    IF NOT _AxisReference^.Inputs.DriveStatusWord_S_0_0135_0_0.ReadyForOperationBit0 OR NOT _AxisReference^.Inputs.DriveStatusWord_S_0_0135_0_0.ReadyForOperationBit1 THEN
                        _State := UINT#388;
                    ELSIF _AxisReference^.Inputs.DriveStatusWord_S_0_0135_0_0.DriveErrorZKL1 OR
                        (_AxisReference^.Inputs.DriveStatusWord_S_0_0135_0_0.WarningZKL2
                        AND _AxisReference^.Inputs.DiagnosticMessage_S_0_0390_0_0 >= DWORD#16#C00E0000) THEN
                        IF MC_MoveVelocityErrorID = DINT#0 THEN
                            MC_MoveVelocityErrorID := TO_DINT(_AxisReference^.Inputs.DiagnosticMessage_S_0_0390_0_0 AND DWORD#16#000FFFFF);
                        END_IF;
                        _State := UINT#389;
                    ELSIF _AxisReference^.Data.Cycle <> MC_MoveVelocityCycle THEN
                        _AxisReference^.Data.Cycle := _AxisReference^.Data.Cycle - ULINT#1;
                        _State := UINT#388;
                    END_IF;
                END_IF;

                THIS.CallTimers(TRUE,FALSE);
                THIS.AxoMoveVelocity_Task.ThrowWhen(_errorTimer.output );
                THIS.AxoMoveVelocity_Task.ThrowWhen(THIS.AxoMoveVelocity_Task.Duration >= DriveConfig.TaskTimeout AND DriveConfig.TaskTimeout > T#0s ,'<#AxoMoveVelocity_Task timeout.#>');
                DriveStatus.Action.Id := _State;
            ELSE
                InVelocity := FALSE;
            END_IF;
            IF THIS.AxoMoveVelocity_Task.DoneReached() AND _State>=UINT#380 AND _State<=UINT#389 THEN
                _AxisReference^.Status.CurrentMotionTaskId := AXOpen.Components.Drives.eAxoMotionTaskId#Axo_Done;
                // _AxisReference^.Outputs.SignalControlWord_S_0_0145_0_0.JogPositive := FALSE;
                // _AxisReference^.Outputs.SignalControlWord_S_0_0145_0_0.JogNegative := FALSE;
                MC_MoveVelocityErrorID := DINT#0;
                _State := UINT#0;
            END_IF;
            IF THIS.AxoMoveVelocity_Task.RestoreTriggered() AND _State>=UINT#380 AND _State<=UINT#389 THEN
                _AxisReference^.Status.CurrentMotionTaskId := AXOpen.Components.Drives.eAxoMotionTaskId#Axo_None;
                // _AxisReference^.Outputs.SignalControlWord_S_0_0145_0_0.JogPositive := FALSE;
                // _AxisReference^.Outputs.SignalControlWord_S_0_0145_0_0.JogNegative := FALSE;
                MC_MoveVelocityErrorID := DINT#0;
                _State := UINT#0;
                MC_MoveVelocityCycle := ULINT#0;
            END_IF;
            ErrorID := MC_MoveVelocityErrorID;
            MC_MoveVelocityExecute_PV := Execute;
        END_METHOD

        ///<summary>
        /// This method continuously exerts a torque or force of the specified magnitude. This magnitude is
        /// approached using a defined ramp (‘TorqueRamp’), and the method sets the ‘InTorque’ output if the
        /// commanded torque level is reached. This method is applicable for force and torque. When there is no external
        /// load, force is applicable. Positive torque is in the positive direction of velocity.
        ///</summary>
        VAR INTERNAL
            MC_TorqueControlExecute_PV					: 	BOOL;				//Execute - previous value
            MC_TorqueControlErrorID					    : 	DINT;
            MC_TorqueControlCycle					    : 	ULINT;
            MC_TorqueControlContinuousUpdate_SV         :   BOOL;
            MC_TorqueControlTorque_PV                   :   LREAL;
            MC_TorqueControlTorqueRamp_PV               :   LREAL;
            MC_TorqueControlPositionLimit_PV            :   LREAL;
            MC_TorqueControlVelocity_PV                 :   LREAL;
            MC_TorqueControlAcceleration_PV             :   LREAL;
            MC_TorqueControlDeceleration_PV             :   LREAL;
            MC_TorqueControlJerk_PV                     :   LREAL;
            MC_TorqueControlDirection_PV                :   AXOpen.Components.Abstractions.Drives.eAxoDriveDirection;
        END_VAR
        METHOD PUBLIC OVERRIDE MC_TorqueControl
            VAR_INPUT
                AxisRef         :   AXOpen.Components.Abstractions.Drives.IAxoAxisReference;
                Execute         :   BOOL;                       //  Start the motion at rising edge
                ContinuousUpdate:   BOOL;                       //  Activate ‘ContinuousUpdate’ - target parameters should be changed during movement
                Torque          :   LREAL;                      //  Value of the torque (Torque or force in technical unit [u])
                TorqueRamp      :   LREAL;                      //  The maximum time derivative of the set value of the torque or force (in technical unit per sec. [u/s])
                PositionLimit   :   LREAL;                      //  Position limit
                Velocity        :   LREAL;                      //  Absolute value of the maximum velocity.
                Acceleration    :   LREAL;                      //  Value of the maximum acceleration (acceleration is applicable with same sign of torque and velocity)
                Deceleration    :   LREAL;                      //  Value of the maximum deceleration (deceleration is applicable with opposite signs of torque and velocity)
                Jerk            :   LREAL;                      //  Value of the maximum jerk
                Direction       :   AXOpen.Components.Abstractions.Drives.eAxoDriveDirection;         //  Enum type (1 of 2 values: PositiveDirection, NegativeDirection or CurrentDirection). Specifies the direction of the torque. (Note: Torque input can be signed value).
            END_VAR
            VAR_OUTPUT
                InTorque        :   BOOL;                       //  Setpoint value of torque or force equals the commandedvalue
                Busy            :   BOOL;                       //  The method is not finished and new output values are to be expected
                Active          :   BOOL;                       //  Indicates that the method has control on the axis
                CommandAborted  :   BOOL;                       //  ‘Command’ is aborted by another command
                Error           :   BOOL;                       //  Signals that an error has occurred within the method
                ErrorID         :   DINT;                       //  Error identification
            END_VAR
            VAR
                _AxisReference          :   REF_TO AxoCtrlxDriveXscAxisReference;
                Torque_                 :   LREAL;
                PositiveDirection_      :   BOOL;
                TorqueWindowPerCent     :   LREAL := LREAL#5.0;
                TorqueWindowMin         :   LREAL;
                TorqueWindowMax         :   LREAL;
            END_VAR

            _AxisReference ?= AxisRef;

            IF(_AxisReference = NULL) THEN
                Messenger.Activate(     UINT#1530, eAxoMessageCategory#ProgrammingError);
                DriveStatus.Error.Id := UINT#1530;
                RETURN;
            END_IF;

            IF THIS.AxoTorqueControl_Task.StartTriggered()  THEN
                _AxisReference^.Status.CurrentMotionTaskId := AXOpen.Components.Drives.eAxoMotionTaskId#Axo_TorqueControl;
            END_IF;

            IF Execute AND NOT MC_TorqueControlExecute_PV AND _State = UINT#0 THEN
                _AxisReference^.Data.Cycle := _AxisReference^.Data.Cycle + ULINT#2;
                MC_TorqueControlCycle := _AxisReference^.Data.Cycle ;
            END_IF;

            IF Execute THEN
                Messenger.ActivateOnCondition(ULINT#1531,Direction <> AXOpen.Components.Abstractions.Drives.eAxoDriveDirection#PositiveDirection AND Direction <> AXOpen.Components.Abstractions.Drives.eAxoDriveDirection#NegativeDirection, eAxoMessageCategory#ProgrammingError);
                Messenger.ActivateOnCondition(ULINT#1532, Execute AND Velocity <= 0, eAxoMessageCategory#ProgrammingError);
                Messenger.ActivateOnCondition(ULINT#1533, Execute AND Acceleration <= 0, eAxoMessageCategory#ProgrammingError);
                Messenger.ActivateOnCondition(ULINT#1534, Execute AND Deceleration <= 0, eAxoMessageCategory#ProgrammingError);
                Messenger.ActivateOnCondition(ULINT#1535, Execute AND Jerk <= 0, eAxoMessageCategory#ProgrammingError);
                Messenger.ActivateOnCondition(ULINT#1536, Execute AND Torque = 0, eAxoMessageCategory#ProgrammingError);
                Messenger.ActivateOnCondition(ULINT#1537, Execute AND TorqueRamp <= 0, eAxoMessageCategory#ProgrammingError);

                IF Direction = AXOpen.Components.Abstractions.Drives.eAxoDriveDirection#PositiveDirection THEN
                    Torque_ := Torque;
                ELSIF Direction = AXOpen.Components.Abstractions.Drives.eAxoDriveDirection#NegativeDirection THEN
                    Torque_ := -1 * Torque;
                ELSE
                    RETURN;
                END_IF;
                PositiveDirection_ := Torque_ > 0;

                IF NOT ContinuousUpdate THEN
                    MC_TorqueControlContinuousUpdate_SV := FALSE;
                END_IF;

                IF _State = UINT#0 THEN
                    Busy := TRUE;
                    Active := TRUE;
                    MC_TorqueControlErrorID := DINT#0;
                    // _AxisReference^.Outputs.DriveControlWord_S_0_0134_0_0.DriveHalt := FALSE;
                    // _AxisReference^.Outputs.DriveControlWord_S_0_0134_0_0.DriveEnable := FALSE;
                    // _AxisReference^.Outputs.DriveControlWord_S_0_0134_0_0.DriveOn := FALSE;
                    // _AxisReference^.Outputs.SignalControlWord_S_0_0145_0_0.AcceptanceOfPositioningCommandValue := FALSE;
                    _AxisReference^.Outputs.SignalControlWord_S_0_0145_0_0.HomingControl := FALSE;
                    _AxisReference^.Outputs.SignalControlWord_S_0_0145_0_0.AbsoluteRelative := FALSE;
                    _AxisReference^.Outputs.SignalControlWord_S_0_0145_0_0.ImmediateChange := FALSE;
                    _AxisReference^.Outputs.SignalControlWord_S_0_0145_0_0.ClearError := FALSE;
                    _AxisReference^.Outputs.SignalControlWord_S_0_0145_0_0.JogPositive := FALSE;
                    _AxisReference^.Outputs.SignalControlWord_S_0_0145_0_0.JogNegative := FALSE;
                    _AxisReference^.Outputs.SignalControlWord_S_0_0145_0_0.SwitchToCM := FALSE;
                    _AxisReference^.Outputs.SignalControlWord_S_0_0145_0_0.SwitchTo0M := TRUE;
                    // _AxisReference^.Outputs.SignalControlWord_S_0_0145_0_0.CancelReferencePoint := FALSE;
                    // _AxisReference^.Outputs.SignalControlWord_S_0_0145_0_0.SetAbsPositionFunction := FALSE;
                    MC_TorqueControlContinuousUpdate_SV := ContinuousUpdate;
                    _State := UINT#390;
                    THIS.CallTimers(FALSE);
                END_IF;
                IF _State = UINT#390 THEN
                    Busy := TRUE;
                    Active := TRUE;
                    IF Velocity > 0 AND Acceleration > 0 AND Deceleration > 0 AND Jerk > 0 AND Torque <> 0 AND TorqueRamp > 0 THEN
                        _AxisReference^.Outputs.CommandTorque_S_0_0080_0_0          :=  TO_INT(Torque_          *   ScalingConstantRequiredTorque);
                        _AxisReference^.Outputs.CommandPosition_S_0_0282_0_0        :=  TO_DINT(PositionLimit   *   ScalingConstantRequiredPosition);
                        _AxisReference^.Outputs.CommandVelocity_S_0_0259_0_0        :=  TO_DINT(Velocity        *   ScalingConstantRequiredVelocity     *   _AxisReference^.Data.OverrideVelocityFactor);
                        _AxisReference^.Outputs.CommandAcceleration_S_0_0260_0_0    :=  TO_DINT(Acceleration    *   ScalingConstantRequiredAcceleration *   _AxisReference^.Data.OverrideAccelerationFactor);
                        _AxisReference^.Outputs.CommandDecceleration_S_0_0359_0_0   :=  TO_DINT(Deceleration    *   ScalingConstantRequiredDeceleration *   _AxisReference^.Data.OverrideAccelerationFactor);
                        _AxisReference^.Outputs.CommandJerk_S_0_0193_0_0            :=  TO_DINT(Jerk            *   ScalingConstantRequiredJerk         *   _AxisReference^.Data.OverrideJerkFactor);

                        MC_TorqueControlPositionLimit_PV :=  PositionLimit;
                        MC_TorqueControlVelocity_PV      :=  Velocity;
                        MC_TorqueControlAcceleration_PV  :=  Acceleration;
                        MC_TorqueControlDeceleration_PV  :=  Deceleration;
                        MC_TorqueControlJerk_PV          :=  Jerk;
                        MC_TorqueControlDirection_PV     :=  Direction;
                        MC_TorqueControlTorque_PV        :=  Torque;
                        MC_TorqueControlTorqueRamp_PV    :=  TorqueRamp;
                        IF PositiveDirection_ AND THIS.ActualPosition >= MC_TorqueControlPositionLimit_PV THEN
                            _State := UINT#399;
                            THIS.CallTimers(FALSE);
                            Messenger.Activate(         UINT#1538, eAxoMessageCategory#ProgrammingError);
                            MC_TorqueControlErrorID :=  DINT#1538;
                        ELSIF NOT PositiveDirection_ AND THIS.ActualPosition <= MC_TorqueControlPositionLimit_PV THEN
                            _State := UINT#399;
                            THIS.CallTimers(FALSE);
                            Messenger.Activate(         UINT#1539, eAxoMessageCategory#ProgrammingError);
                            MC_TorqueControlErrorID :=  DINT#1539;
                        ELSE
                            _State := UINT#391;
                            THIS.CallTimers(FALSE);
                        END_IF;
                    END_IF;
                END_IF;
                //Writing Torque/force control: Ramp value (0x2838:01 / S-0-0822 / --)
                IF _State = UINT#391 THEN
                    IF _infoTimer.output THEN
                        TaskMessenger.Activate( UINT#591, eAxoMessageCategory#Potential);
                        DriveStatus.Error.Id := UINT#591;
                    END_IF;
                    Busy := TRUE;
                    Active := TRUE;
                    _word :=  TO_WORD(TO_INT(TorqueRamp * ScalingConstantRequiredTorque));
                    _data2[0] := _word.%B0;
                    _data2[1] := _word.%B1;
                    _WriteRecord(   request     :=  TRUE,
                                    hardwareID  :=  (AxisRefExt.HWIDs.HW_S_0_0134_0_0),
                                    index       :=  DINT#822,
                                    length      :=  UINT#2,
                                    record      :=  _data2);
                    IF NOT _WriteRecord.busy AND _WriteRecord.done AND NOT _WriteRecord.error THEN
                        _WriteRecord(request := FALSE, record := _data2);
                        _State := UINT#392;
                        THIS.CallTimers(FALSE);
                    ElSIF _WriteRecord.error THEN
                        _WriteRecord(request := FALSE, record := _data2);
                        Messenger.Activate(             UINT#1540, eAxoMessageCategory#Error);
                        MC_WriteRealParameterErrorID := WORD#1540;
                        _State := UINT#399;
                        THIS.CallTimers(FALSE);
                    END_IF;
                END_IF;
                //Writing Torque/force control: Ramp time (0x2838:02 / S-0-0823 / --)
                IF _State = UINT#392 THEN
                    IF _infoTimer.output THEN
                        TaskMessenger.Activate( UINT#592, eAxoMessageCategory#Potential);
                        DriveStatus.Error.Id := UINT#592;
                    END_IF;
                    Busy := TRUE;
                    Active := TRUE;
                    _word :=  TO_WORD(TO_UINT(AxoTorqueControl_TorqueRampTime * ScalingConstantRequiredTorqueRampTime)); // value * 10, Max 65535.5 ms
                    _data2[0] := _word.%B0;
                    _data2[1] := _word.%B1;
                    _WriteRecord(   request     :=  TRUE,
                                    hardwareID  :=  (AxisRefExt.HWIDs.HW_S_0_0134_0_0),
                                    index       :=  DINT#823,
                                    length      :=  UINT#2,
                                    record      :=  _data2);
                    IF NOT _WriteRecord.busy AND _WriteRecord.done AND NOT _WriteRecord.error THEN
                        _WriteRecord(request := FALSE, record := _data2);
                        _State := UINT#393;
                        THIS.CallTimers(FALSE);
                    ElSIF _WriteRecord.error THEN
                        _WriteRecord(request := FALSE, record := _data2);
                        Messenger.Activate(             UINT#1541, eAxoMessageCategory#Error);
                        MC_WriteRealParameterErrorID := WORD#1541;
                        _State := UINT#399;
                        THIS.CallTimers(FALSE);
                    END_IF;
                END_IF;
                //Writing Torque/force control: High velocity limit value (0x60C9:00 / P-0-0421.0.3 / P-0-2249)
                IF _State = UINT#393 THEN
                    IF _infoTimer.output THEN
                        TaskMessenger.Activate( UINT#593, eAxoMessageCategory#Potential);
                        DriveStatus.Error.Id := UINT#593;
                    END_IF;
                    Busy := TRUE;
                    Active := TRUE;
                    _dword :=  TO_DWORD(TO_DINT(ABS(Velocity) * ScalingConstantRequiredVelocity * _AxisReference^.Data.OverrideVelocityFactor));
                    _data4[0] := _dword.%B0;
                    _data4[1] := _dword.%B1;
                    _data4[2] := _dword.%B2;
                    _data4[3] := _dword.%B3;
                    _WriteRecord(   request     :=  TRUE,
                                    hardwareID  :=  (AxisRefExt.HWIDs.HW_S_0_0134_0_0),
                                    index       :=  DINT#6345,
                                    length      :=  UINT#4,
                                    record      :=  _data4);
                    IF NOT _WriteRecord.busy AND _WriteRecord.done AND NOT _WriteRecord.error THEN
                        _WriteRecord(request := FALSE, record := _data4);
                        _State := UINT#394;
                        THIS.CallTimers(FALSE);
                    ElSIF _WriteRecord.error THEN
                        _WriteRecord(request := FALSE, record := _data4);
                        Messenger.Activate(             UINT#1542, eAxoMessageCategory#Error);
                        MC_WriteRealParameterErrorID := WORD#1542;
                        _State := UINT#399;
                        THIS.CallTimers(FALSE);
                    END_IF;
                END_IF;
                //Writing Torque/force control: Low velocity limit value (0x60C8:00 / P-0-0421.0.4 / P-0-2250)
                IF _State = UINT#394 THEN
                    IF _infoTimer.output THEN
                        TaskMessenger.Activate( UINT#594, eAxoMessageCategory#Potential);
                        DriveStatus.Error.Id := UINT#594;
                    END_IF;
                    Busy := TRUE;
                    Active := TRUE;
                    _dword :=  TO_DWORD(TO_DINT(-1.0 * ABS(Velocity) * ScalingConstantRequiredVelocity * _AxisReference^.Data.OverrideVelocityFactor));
                    _data4[0] := _dword.%B0;
                    _data4[1] := _dword.%B1;
                    _data4[2] := _dword.%B2;
                    _data4[3] := _dword.%B3;
                    _WriteRecord(   request     :=  TRUE,
                                    hardwareID  :=  (AxisRefExt.HWIDs.HW_S_0_0134_0_0),
                                    index       :=  DINT#6346,
                                    length      :=  UINT#4,
                                    record      :=  _data4);
                    IF NOT _WriteRecord.busy AND _WriteRecord.done AND NOT _WriteRecord.error THEN
                        _WriteRecord(request := FALSE, record := _data4);
                        _State := UINT#395;
                        THIS.CallTimers(FALSE);
                    ElSIF _WriteRecord.error THEN
                        _WriteRecord(request := FALSE, record := _data4);
                        Messenger.Activate(             UINT#1543, eAxoMessageCategory#Error);
                        MC_WriteRealParameterErrorID := WORD#1543;
                        _State := UINT#399;
                        THIS.CallTimers(FALSE);
                    END_IF;
                END_IF;
                //Executing movement
                IF _State = UINT#395 THEN
                    IF _infoTimer.output THEN
                        TaskMessenger.Activate( UINT#595, eAxoMessageCategory#Potential);
                        DriveStatus.Error.Id := UINT#595;
                    END_IF;
                    Busy := TRUE;
                    Active := TRUE;
                    _AxisReference^.Outputs.DriveControlWord_S_0_0134_0_0.DriveHalt := TRUE;
                    _AxisReference^.Outputs.DriveControlWord_S_0_0134_0_0.CommandOperationModeBit0 := TRUE; // torque with velocity limit
                    _AxisReference^.Outputs.DriveControlWord_S_0_0134_0_0.CommandOperationModeBit1 := FALSE;
                    _AxisReference^.Outputs.DriveControlWord_S_0_0134_0_0.CommandOperationModeBit2 := FALSE;
                    // IF      _AxisReference^.Inputs.DriveStatusWord_S_0_0135_0_0.ActualOperatingModeBit0 AND
                    //     NOT _AxisReference^.Inputs.DriveStatusWord_S_0_0135_0_0.ActualOperatingModeBit1 AND
                    //     NOT _AxisReference^.Inputs.DriveStatusWord_S_0_0135_0_0.ActualOperatingModeBit2 THEN
                    IF      _AxisReference^.Inputs.DriveStatusWord_S_0_0135_0_0.ActualOperatingModeBit0 AND
                        NOT _AxisReference^.Inputs.DriveStatusWord_S_0_0135_0_0.ActualOperatingModeBit1 AND
                        NOT _AxisReference^.Inputs.DriveStatusWord_S_0_0135_0_0.ActualOperatingModeBit2 AND
                            _AxisReference^.Inputs.DriveStatusWord_S_0_0135_0_0.CommandProcessingStatus AND
                        NOT _AxisReference^.Inputs.DriveStatusWord_S_0_0135_0_0.InStandstill  THEN
                        _State := UINT#396;
                        THIS.CallTimers(FALSE);
                    END_IF;
                END_IF;
                IF PositiveDirection_  THEN
                    TorqueWindowMax := Torque_ + (Torque_ * TorqueWindowPerCent / REAL#100.0);
                    TorqueWindowMin := Torque_ - (Torque_ * TorqueWindowPerCent / REAL#100.0);
                ELSE
                    TorqueWindowMax := Torque_ - (Torque_ * TorqueWindowPerCent / REAL#100.0);
                    TorqueWindowMin := Torque_ + (Torque_ * TorqueWindowPerCent / REAL#100.0);
                END_IF;
                InTorque := ActualTorque >= TorqueWindowMin AND ActualTorque <= TorqueWindowMax;
                IF _State = UINT#396 THEN
                    IF InTorque AND NOT MC_TorqueControlContinuousUpdate_SV THEN
                        _State := UINT#397;
                        THIS.CallTimers(FALSE);
                    END_IF;
                END_IF;
                IF _State = UINT#397 THEN
                    MC_TorqueControlCycle := ULINT#0;
                END_IF;
                IF _State = UINT#398 THEN
                    CommandAborted := TRUE; // AxoTorqueControl_Task will be aborted in AxoDrive
                END_IF;
                IF _State = UINT#399 THEN
                    MC_TorqueControlCycle := ULINT#0;
                    Error := TRUE;     // AxoTorqueControl_Task will pass to error in AxoDrive
                END_IF;

                IF (_State>=UINT#395 AND _State <= UINT#397) THEN
                    IF  (    PositiveDirection_ AND ActualPosition > PositionLimit) OR
                        (NOT PositiveDirection_ AND ActualPosition < PositionLimit) THEN
                        Messenger.Activate(         UINT#1542, eAxoMessageCategory#ProgrammingError);
                        MC_TorqueControlErrorID :=  DINT#1542;
                        _AxisReference^.Outputs.DriveControlWord_S_0_0134_0_0.DriveHalt := FALSE;
                        _State := UINT#399;
                    END_IF;
                END_IF;

                IF _State>=UINT#390 AND _State<UINT#397 THEN
                    IF MC_TorqueControlContinuousUpdate_SV AND (
                        MC_TorqueControlTorque_PV        <>  Torque OR
                        MC_TorqueControlTorqueRamp_PV    <>  TorqueRamp OR
                        MC_TorqueControlPositionLimit_PV <>  PositionLimit OR
                        MC_TorqueControlVelocity_PV      <>  Velocity OR
                        MC_TorqueControlAcceleration_PV  <>  Acceleration OR
                        MC_TorqueControlDeceleration_PV  <>  Deceleration OR
                        MC_TorqueControlJerk_PV          <>  Jerk OR
                        MC_TorqueControlDirection_PV     <>  Direction ) THEN
                        IF TRUE THEN
                            _State := UINT#390;
                        END_IF;
                    END_IF;
                    IF NOT _AxisReference^.Inputs.DriveStatusWord_S_0_0135_0_0.ReadyForOperationBit0 OR NOT _AxisReference^.Inputs.DriveStatusWord_S_0_0135_0_0.ReadyForOperationBit1 THEN
                        _State := UINT#398;
                    ELSIF _AxisReference^.Inputs.DriveStatusWord_S_0_0135_0_0.DriveErrorZKL1 OR
                        (_AxisReference^.Inputs.DriveStatusWord_S_0_0135_0_0.WarningZKL2 AND _AxisReference^.Inputs.DiagnosticMessage_S_0_0390_0_0 >= DWORD#16#C00E0000) THEN
                        IF MC_TorqueControlErrorID = DINT#0 THEN
                            MC_TorqueControlErrorID := TO_DINT(_AxisReference^.Inputs.DiagnosticMessage_S_0_0390_0_0 AND DWORD#16#000FFFFF);
                        END_IF;
                        _State := UINT#399;
                    ELSIF _AxisReference^.Data.Cycle <> MC_TorqueControlCycle THEN
                        _AxisReference^.Data.Cycle := _AxisReference^.Data.Cycle - ULINT#1;
                        _State := UINT#398;
                    END_IF;
                END_IF;
            ELSE
                InTorque := FALSE;
            END_IF;

            IF THIS.AxoTorqueControl_Task.DoneReached() AND _State>=UINT#390 AND _State<=UINT#399 THEN
                _AxisReference^.Status.CurrentMotionTaskId := AXOpen.Components.Drives.eAxoMotionTaskId#Axo_Done;
                MC_TorqueControlErrorID := DINT#0;
                // MC_TorqueControlCycle := ULINT#0;
                _State := UINT#0;
            END_IF;

            IF THIS.AxoTorqueControl_Task.RestoreTriggered() AND _State>=UINT#390 AND _State<=UINT#399 THEN
                _AxisReference^.Status.CurrentMotionTaskId := AXOpen.Components.Drives.eAxoMotionTaskId#Axo_None;
                MC_TorqueControlErrorID := DINT#0;
                MC_TorqueControlCycle := ULINT#0;
                _State := UINT#0;
            END_IF;

            ErrorID := MC_TorqueControlErrorID;
            MC_TorqueControlExecute_PV := Execute;
        END_METHOD

        ///<summary>
        /// This method shifts the coordinate system of an axis by manipulating both the set-point position as well as the
        /// actual position of an axis with the same value without any movement caused. (Re-calibration with same following error).
        /// This can be used for instance for a reference situation. This method can also be used during motion without changing
        /// the commanded position, which is now positioned in the shifted coordinate system.
        ///</summary>
        VAR INTERNAL
            MC_SetPositionExecute_PV				: 	BOOL;				//Execute - previous value
            MC_SetPositionErrorID					: 	DINT;
            MC_SetPositionCycle					    : 	ULINT;
            MC_SetPositionActualPosition            : 	LINT;
            MC_SetPositionPowerStatusPV             : 	BOOL;
        END_VAR
        METHOD PUBLIC OVERRIDE MC_SetPosition
            VAR_INPUT
                AxisRef         :   AXOpen.Components.Abstractions.Drives.IAxoAxisReference;
                Execute         :   BOOL;                       //  Start setting position in axis
                Position        :   LREAL;                       //  Position unit [u] (Means ‘Distance’ if ‘Relative’= TRUE)
                Relative        :   BOOL;                       //  ‘Relative’ distance if True, ‘Absolute’ position if False (= Default)
                ExecutionMode   :   AXOpen.Components.Abstractions.Drives.eAxoExecutionMode;          //  Defines the chronological sequence of the method.
            END_VAR
            VAR_OUTPUT
                Done            :   BOOL;                       //  ‘Position’ has new value
                Busy            :   BOOL;                       //  The method is not finished and new output values are to be expected
                Error           :   BOOL;                       //  Signals that an error has occurred within the method
                ErrorID         :   DINT;                       //  Error identification
            END_VAR
            VAR
                _AxisReference :  REF_TO AxoCtrlxDriveXscAxisReference;
            END_VAR

            _AxisReference ?= AxisRef;

            IF(_AxisReference = NULL) THEN
                Messenger.Activate(     UINT#1550, eAxoMessageCategory#ProgrammingError);
                DriveStatus.Error.Id := UINT#1550;
                RETURN;
            END_IF;

            IF THIS.AxoSetPosition_Task.StartTriggered() THEN
                _AxisReference^.Status.CurrentMotionTaskId := AXOpen.Components.Drives.eAxoMotionTaskId#Axo_SetPosition;
            END_IF;

            IF Execute AND NOT MC_SetPositionExecute_PV AND _State = UINT#0 THEN
                _AxisReference^.Data.Cycle := _AxisReference^.Data.Cycle + ULINT#2;
                MC_SetPositionCycle := _AxisReference^.Data.Cycle ;
            END_IF;

            IF Execute THEN
                IF _State = UINT#0 THEN
                    Busy := TRUE;
                    MC_SetPositionErrorID := DINT#0;
                    DriveStatus.Error.Id :=  UINT#0;
                    TaskMessenger.Restore();
                    THIS.CallTimers(FALSE);
                    // _AxisReference^.Outputs.DriveControlWord_S_0_0134_0_0.IPOSYNC := FALSE;
                    // _AxisReference^.Outputs.DriveControlWord_S_0_0134_0_0.DriveHalt := FALSE;
                    // _AxisReference^.Outputs.DriveControlWord_S_0_0134_0_0.DriveEnable := FALSE;
                    // _AxisReference^.Outputs.DriveControlWord_S_0_0134_0_0.DriveOn := FALSE;
                    _AxisReference^.Outputs.SignalControlWord_S_0_0145_0_0.AcceptanceOfPositioningCommandValue := FALSE;
                    _AxisReference^.Outputs.SignalControlWord_S_0_0145_0_0.HomingControl := FALSE;
                    _AxisReference^.Outputs.SignalControlWord_S_0_0145_0_0.AbsoluteRelative := FALSE;
                    _AxisReference^.Outputs.SignalControlWord_S_0_0145_0_0.ImmediateChange := FALSE;
                    _AxisReference^.Outputs.SignalControlWord_S_0_0145_0_0.JogPositive := FALSE;
                    _AxisReference^.Outputs.SignalControlWord_S_0_0145_0_0.JogNegative := FALSE;
                    _AxisReference^.Outputs.SignalControlWord_S_0_0145_0_0.ClearError := FALSE;
                    MC_SetPositionPowerStatusPV := _AxisReference^.Inputs.DriveStatusWord_S_0_0135_0_0.ReadyForOperationBit1 AND _AxisReference^.Inputs.DriveStatusWord_S_0_0135_0_0.ReadyForOperationBit0;
                    _State := UINT#400;
                    THIS.CallTimers(FALSE);
                END_IF;
                // Power off
                IF _State = UINT#400 THEN
                    IF _infoTimer.output THEN
                        TaskMessenger.Activate( UINT#600, eAxoMessageCategory#Potential);
                        DriveStatus.Error.Id := UINT#600;
                    END_IF;
                    Busy := TRUE;
                    _AxisReference^.Outputs.DriveControlWord_S_0_0134_0_0.DriveHalt := FALSE;
                    _AxisReference^.Outputs.DriveControlWord_S_0_0134_0_0.DriveEnable := FALSE;
                    _AxisReference^.Outputs.DriveControlWord_S_0_0134_0_0.DriveOn := FALSE;
                    IF NOT _AxisReference^.Inputs.DriveStatusWord_S_0_0135_0_0.ReadyForOperationBit0 THEN
                        _State := UINT#401;
                        THIS.CallTimers(FALSE);
                        RETURN;
                    END_IF;
                END_IF;
                // Reseting InReference flag
                IF _State = UINT#401 THEN
                    IF _infoTimer.output THEN
                        TaskMessenger.Activate( UINT#601, eAxoMessageCategory#Potential);
                        DriveStatus.Error.Id := UINT#601;
                    END_IF;
                    Busy := TRUE;
                    _AxisReference^.Outputs.SignalControlWord_S_0_0145_0_0.CancelReferencePoint := TRUE;
                    IF NOT _AxisReference^.Inputs.DriveStatusWord_S_0_0135_0_0.InReference THEN
                        _AxisReference^.Outputs.SignalControlWord_S_0_0145_0_0.CancelReferencePoint := FALSE;
                        _State := UINT#402;
                        THIS.CallTimers(FALSE);
                        RETURN;
                    END_IF;
                END_IF;
                //Writing Homing configuration ENC_1: Home offset (0x607C:00 / S-0-0052 / --)
                IF _State = UINT#402 THEN
                    IF _infoTimer.output THEN
                        TaskMessenger.Activate( UINT#602, eAxoMessageCategory#Potential);
                        DriveStatus.Error.Id := UINT#602;
                    END_IF;
                    Busy := TRUE;
                    _dword :=  TO_DWORD(TO_DINT(Position * ScalingConstantRequiredPosition));
                    _data4[0] := _dword.%B0;
                    _data4[1] := _dword.%B1;
                    _data4[2] := _dword.%B2;
                    _data4[3] := _dword.%B3;
                    _WriteRecord(   request     :=  TRUE,
                                    hardwareID  :=  (AxisRefExt.HWIDs.HW_S_0_0134_0_0),
                                    index       :=  DINT#52,
                                    length      :=  UINT#4,
                                    record      :=  _data4);
                    IF NOT _WriteRecord.busy AND _WriteRecord.done AND NOT _WriteRecord.error THEN
                        _State := UINT#403;
                        THIS.CallTimers(FALSE);
                    ElSIF _WriteRecord.error THEN
                        Messenger.Activate( UINT#1551, eAxoMessageCategory#Error);
                        MC_HomeErrorID :=   DINT#1551;
                        _WriteRecord(request := FALSE, record := _data4);
                        _State := UINT#409;
                        THIS.CallTimers(FALSE);
                    END_IF;
                END_IF;
                IF _State = UINT#403 THEN
                    IF _infoTimer.output THEN
                        TaskMessenger.Activate( UINT#603, eAxoMessageCategory#Potential);
                        DriveStatus.Error.Id := UINT#603;
                    END_IF;
                    Busy := TRUE;
                    _WriteRecord(request := FALSE, record := _data4);
                    IF NOT _WriteRecord.busy AND NOT _WriteRecord.done AND NOT _WriteRecord.error  THEN
                        _State := UINT#404;
                        THIS.CallTimers(FALSE);
                    END_IF;
                END_IF;
                IF _State = UINT#404 THEN
                    IF _infoTimer.output THEN
                        TaskMessenger.Activate( UINT#604, eAxoMessageCategory#Potential);
                        DriveStatus.Error.Id := UINT#604;
                    END_IF;
                    Busy := TRUE;
                    _AxisReference^.Outputs.SignalControlWord_S_0_0145_0_0.SetAbsPositionFunction := TRUE;
                    IF _AxisReference^.Inputs.DriveStatusWord_S_0_0135_0_0.InReference THEN
                        _AxisReference^.Outputs.SignalControlWord_S_0_0145_0_0.SetAbsPositionFunction := FALSE;
                        IF MC_SetPositionPowerStatusPV THEN
                            _State := UINT#405;
                            THIS.CallTimers(FALSE);
                        ELSE
                            _State := UINT#407;
                            THIS.CallTimers(FALSE);
                        END_IF;
                    END_IF;
                END_IF;
                IF _State = UINT#405 THEN
                    IF _infoTimer.output THEN
                        TaskMessenger.Activate( UINT#605, eAxoMessageCategory#Potential);
                        DriveStatus.Error.Id := UINT#605;
                    END_IF;
                    Busy := TRUE;
                    _AxisReference^.Outputs.DriveControlWord_S_0_0134_0_0.DriveEnable := TRUE;
                    _AxisReference^.Outputs.DriveControlWord_S_0_0134_0_0.DriveOn := TRUE;
                    IF _AxisReference^.Inputs.DriveStatusWord_S_0_0135_0_0.ReadyForOperationBit0 AND _AxisReference^.Inputs.DriveStatusWord_S_0_0135_0_0.ReadyForOperationBit1 THEN
                        _AxisReference^.Outputs.SignalControlWord_S_0_0145_0_0.SetAbsPositionFunction := FALSE;
                        _State := UINT#407;
                        THIS.CallTimers(FALSE);
                    END_IF;
                END_IF;
                IF _State = UINT#407 THEN
                    Done := TRUE;
                    MC_SetPositionCycle := ULINT#0;
                    _AxisReference^.Outputs.SignalControlWord_S_0_0145_0_0.SetAbsPositionFunction := FALSE;
                    _AxisReference^.Outputs.SignalControlWord_S_0_0145_0_0.CancelReferencePoint := FALSE;
                    _AxisReference^.Outputs.SignalControlWord_S_0_0145_0_0.HomingControl := FALSE;
                END_IF;
                IF _State = UINT#408 THEN
                    _AxisReference^.Outputs.SignalControlWord_S_0_0145_0_0.SetAbsPositionFunction := FALSE;
                    _AxisReference^.Outputs.SignalControlWord_S_0_0145_0_0.CancelReferencePoint := FALSE;
                    _AxisReference^.Outputs.SignalControlWord_S_0_0145_0_0.HomingControl := FALSE;
                    MC_SetPositionCycle := ULINT#0;
                    AxoSetPosition_Task.Abort();
                END_IF;
                IF _State = UINT#409 THEN
                    _AxisReference^.Outputs.SignalControlWord_S_0_0145_0_0.SetAbsPositionFunction := FALSE;
                    _AxisReference^.Outputs.SignalControlWord_S_0_0145_0_0.CancelReferencePoint := FALSE;
                    _AxisReference^.Outputs.SignalControlWord_S_0_0145_0_0.HomingControl := FALSE;
                    MC_SetPositionCycle := ULINT#0;
                    AxoSetPosition_Task.ThrowWhen(TRUE);
                    Error := TRUE;
                END_IF;

                IF _State>=UINT#400 AND _State<UINT#407 THEN
                    IF (*NOT _AxisReference^.Inputs.DriveStatusWord_S_0_0135_0_0.ReadyForOperationBit0 OR*) NOT _AxisReference^.Inputs.DriveStatusWord_S_0_0135_0_0.ReadyForOperationBit1 THEN
                        _State := UINT#408;
                    ELSIF _AxisReference^.Inputs.DriveStatusWord_S_0_0135_0_0.DriveErrorZKL1 OR
                        (_AxisReference^.Inputs.DriveStatusWord_S_0_0135_0_0.WarningZKL2 AND _AxisReference^.Inputs.DiagnosticMessage_S_0_0390_0_0 >= DWORD#16#C00E0000) THEN
                        IF MC_SetPositionErrorID = DINT#0 THEN
                            MC_SetPositionErrorID := TO_DINT(_AxisReference^.Inputs.DiagnosticMessage_S_0_0390_0_0 AND DWORD#16#000FFFFF);
                        END_IF;
                        _State := UINT#409;
                    ELSIF _AxisReference^.Data.Cycle <> MC_SetPositionCycle THEN
                        _AxisReference^.Data.Cycle := _AxisReference^.Data.Cycle - ULINT#1;
                        _State := UINT#408;
                    END_IF;
                END_IF;
                THIS.CallTimers(TRUE,FALSE);
                THIS.AxoSetPosition_Task.ThrowWhen(_errorTimer.output );
                THIS.AxoSetPosition_Task.ThrowWhen(THIS.AxoHome_Task.Duration >= DriveConfig.TaskTimeout AND DriveConfig.TaskTimeout > T#0s ,'<#AxoSetPosition_Task timeout.#>');
                DriveStatus.Action.Id := _State;
            END_IF;

            IF THIS.AxoSetPosition_Task.DoneReached() AND _State>=UINT#400 AND _State<=UINT#409 THEN
                _AxisReference^.Status.CurrentMotionTaskId := AXOpen.Components.Drives.eAxoMotionTaskId#Axo_Done;
                MC_SetPositionErrorID := DINT#0;
                _AxisReference^.Outputs.SignalControlWord_S_0_0145_0_0.SetAbsPositionFunction := FALSE;
                _AxisReference^.Outputs.SignalControlWord_S_0_0145_0_0.CancelReferencePoint := FALSE;
                _AxisReference^.Outputs.SignalControlWord_S_0_0145_0_0.HomingControl := FALSE;
                _State := UINT#0;
            END_IF;
            IF THIS.AxoSetPosition_Task.RestoreTriggered() AND _State>=UINT#400 AND _State<=UINT#409 THEN
                _AxisReference^.Status.CurrentMotionTaskId := AXOpen.Components.Drives.eAxoMotionTaskId#Axo_None;
                MC_SetPositionErrorID := DINT#0;
                MC_SetPositionCycle := ULINT#0;
                _AxisReference^.Outputs.SignalControlWord_S_0_0145_0_0.SetAbsPositionFunction := FALSE;
                _AxisReference^.Outputs.SignalControlWord_S_0_0145_0_0.CancelReferencePoint := FALSE;
                _AxisReference^.Outputs.SignalControlWord_S_0_0145_0_0.HomingControl := FALSE;
            _State := UINT#0;
            END_IF;

            ErrorID := MC_SetPositionErrorID;
            MC_SetPositionExecute_PV := Execute;
         END_METHOD

        ///<summary>
        /// This method sets the values of override for the whole axis, and all functions that are working on that axis. The override
        /// parameters contribute as a factor to the calculation of the commanded velocity, acceleration and jerk of the motion.
        ///<summary>
        METHOD PUBLIC OVERRIDE MC_SetOverride
            VAR_INPUT
                AxisRef         :   AXOpen.Components.Abstractions.Drives.IAxoAxisReference;
                Enable          :   BOOL;                       //  If SET, it writes the value of the override factor continuously. If RESET it should keep the last value.
                VelocityFactor  :   LREAL;                      //  New override factor for the velocity
                AccelerationFactor:   LREAL;                    //  New override factor for the acceleration/deceleration
                JerkFactor      :   LREAL;                      //  New override factor for the jer
            END_VAR
            VAR_OUTPUT
                Enabled         :   BOOL;                       //  Signals that the override factor(s) is (are) set successfully
                Busy            :   BOOL;                       //  The method is not finished and new output values are to be expected
                Error           :   BOOL;                       //  Signals that an error has occurred within the method
                ErrorID         :   DINT;                       //  Error identification
            END_VAR
            VAR
                _AxisReference :  REF_TO AxoCtrlxDriveXscAxisReference;
            END_VAR

            _AxisReference ?= AxisRef;

            IF(_AxisReference = NULL) THEN
                Messenger.Activate(     UINT#1570, eAxoMessageCategory#ProgrammingError);
                DriveStatus.Error.Id := UINT#1570;
                RETURN;
            END_IF;

            Messenger.ActivateOnCondition(ULINT#1571, Enable AND  (VelocityFactor <= 0.0 OR  VelocityFactor >= 2.0), eAxoMessageCategory#ProgrammingError);
            Messenger.ActivateOnCondition(ULINT#1572, Enable AND  (AccelerationFactor <= 0.0 OR  AccelerationFactor > 1.0), eAxoMessageCategory#ProgrammingError);
            Messenger.ActivateOnCondition(ULINT#1573, Enable AND  (JerkFactor <= 0.0 OR JerkFactor > 1.0), eAxoMessageCategory#ProgrammingError);
